// TIA Portal V20 export
VAR_GLOBAL   // PLC tag table "SSP1"
   SSP1_Safety1_1 AT %I5250.0 : Bool;
   SSP1_Safety2_1 AT %I5250.1 : Bool;
   SSP1_Safety3_1 AT %I5250.2 : Bool;
   SSP1_Safety4_1 AT %I5250.3 : Bool;
   SSP1_Safety1_2 AT %I5251.0 : Bool;
   SSP1_Safety2_2 AT %I5251.1 : Bool;
   SSP1_Safety3_2 AT %I5251.2 : Bool;
   SSP1_Safety4_2 AT %I5251.3 : Bool;
   SSP1_Valve_Up AT %Q5200.0 : Bool;
   SSP1_Valve_Down AT %Q5200.1 : Bool;
   SSP1_Hydraulic_Unit AT %Q5200.2 : Bool;
   SSP1_Sen_Drv_1 AT %I5200.0 : Bool;
   SSP1_Sen_Drv_2 AT %I5200.1 : Bool;
   SSP1_Sen_Drv_3 AT %I5200.2 : Bool;
   SSP1_Sen_Drv_4 AT %I5200.3 : Bool;
   SSP1_Sen_Val1_Up AT %I5200.4 : Bool;
   SSP1_Sen_Val1_Down AT %I5200.5 : Bool;
   SSP1_Sen_Val2_Up AT %I5200.6 : Bool;
   SSP1_Sen_Val2_Down AT %I5200.7 : Bool;
   SSP1_Hyd_Filtr AT %I5201.0 : Bool;
   SSP1_Hyd_Empty AT %I5201.1 : Bool;
END_VAR
